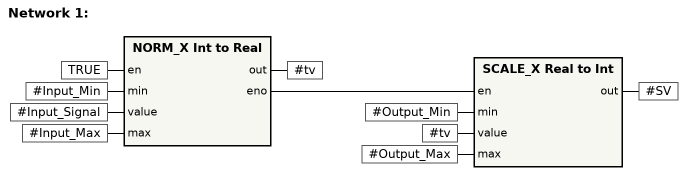
   IF TRUE THEN
       #tv := NORM_X(MIN := #Input_Min, VALUE := #Input_Signal, MAX := #Input_Max);
       #SV := SCALE_X(MIN := #Output_Min, VALUE := #tv, MAX := #Output_Max);
   END_IF;
END_REGION
END_FUNCTION

FUNCTION "CONVERTTIME" : Void   // FC2, FBD
{ S7_Optimized_Access := 'TRUE' }
VERSION : 0.1
   VAR_INPUT
      Int1 : Int;
   END_VAR
   VAR_OUTPUT
      tem1 : Time;
   END_VAR
   VAR_TEMP
      tv : Int;
   END_VAR
BEGIN

REGION Network 1
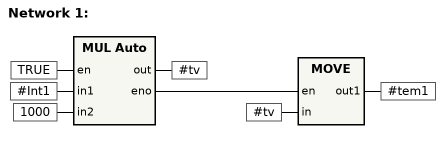
   IF TRUE THEN
       #tv := #Int1 * 1000;
       #tem1 := #tv;
   END_IF;
END_REGION
END_FUNCTION

ORGANIZATION_BLOCK "Main"   // OB1, LAD, ProgramCycle
TITLE = "Main Program Sweep (Cycle)"
{ S7_Optimized_Access := 'TRUE' }
VERSION : 0.1
   VAR_INPUT
      Initial_Call : Bool;   // Initial call of this OB
      Remanence : Bool;   // =True, if remanent data are available
   END_VAR
   VAR_TEMP
      InitiateSequens : Bool;
   END_VAR
   VAR_TEMP   // added for the SCL form of the ladder/FBD networks
      _w1 : Bool;
      _w2 : Bool;
      _w3 : Bool;
      _w4 : Bool;
   END_VAR
BEGIN

REGION Network 1
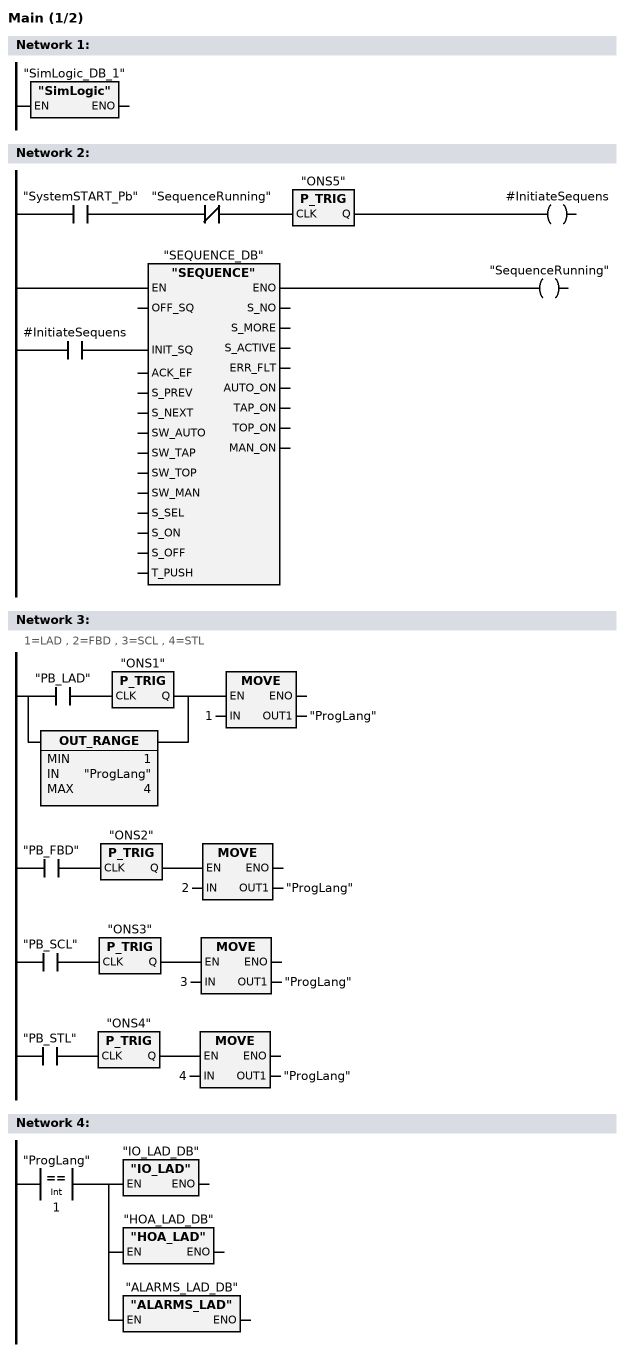
   RUNG wire#powerrail
      "SimLogic_DB_1"()
   END_RUNG
   // the same network as SCL:
   "SimLogic_DB_1"();   // "SimLogic"
END_REGION

REGION Network 2
   RUNG wire#powerrail
      Contact( "SystemSTART_Pb" )
      I_Contact( "SequenceRunning" )
      P_Trig( "ONS5" )
      Coil( #InitiateSequens )
   END_RUNG
   RUNG wire#powerrail
      "SEQUENCE_DB"(INIT_SQ := wire#w1, OFF_SQ :=, ACK_EF :=, S_PREV :=, S_NEXT :=, SW_AUTO :=, SW_TAP :=, SW_TOP :=, SW_MAN :=, S_SEL :=, S_ON :=, S_OFF :=, T_PUSH :=, S_NO =>, S_MORE =>, S_ACTIVE =>, ERR_FLT =>, AUTO_ON =>, TAP_ON =>, TOP_ON =>, MAN_ON =>)
      Coil( "SequenceRunning" )
   END_RUNG
   RUNG wire#powerrail
      Contact( #InitiateSequens )
   END_RUNG wire#w1
   // the same network as SCL:
   #_w1 := "SystemSTART_Pb" AND NOT "SequenceRunning";
   #_w2 := #_w1 AND NOT "ONS5";   // rising edge
   "ONS5" := #_w1;
   #InitiateSequens := #_w2;
   "SEQUENCE_DB"(INIT_SQ := #InitiateSequens, ENO => #_w3);   // "SEQUENCE"
   "SequenceRunning" := #_w3;
END_REGION

REGION Network 3
   // 1=LAD , 2=FBD , 3=SCL , 4=STL
   #_w1 := "PB_LAD" AND NOT "ONS1";   // rising edge
   "ONS1" := "PB_LAD";
   IF #_w1 OR ("ProgLang" < 1) OR ("ProgLang" > 4) THEN "ProgLang" := 1; END_IF;
   #_w2 := "PB_FBD" AND NOT "ONS2";   // rising edge
   "ONS2" := "PB_FBD";
   IF #_w2 THEN "ProgLang" := 2; END_IF;
   #_w3 := "PB_SCL" AND NOT "ONS3";   // rising edge
   "ONS3" := "PB_SCL";
   IF #_w3 THEN "ProgLang" := 3; END_IF;
   #_w4 := "PB_STL" AND NOT "ONS4";   // rising edge
   "ONS4" := "PB_STL";
   IF #_w4 THEN "ProgLang" := 4; END_IF;
END_REGION

REGION Network 4
   RUNG wire#powerrail
      { S7_Templates := "SrcType := Int" } EQ_Contact(in1 := "ProgLang", in2 := 1)
      wire#w1
      "IO_LAD_DB"()
   END_RUNG
   RUNG wire#w1
      "HOA_LAD_DB"()
   END_RUNG
   RUNG wire#w1
      "ALARMS_LAD_DB"()
   END_RUNG
   // the same network as SCL:
   #_w1 := "ProgLang" = 1;
   IF #_w1 THEN
       "IO_LAD_DB"();   // "IO_LAD"
       "HOA_LAD_DB"();   // "HOA_LAD"
       "ALARMS_LAD_DB"();   // "ALARMS_LAD"
   END_IF;
END_REGION

REGION Network 5
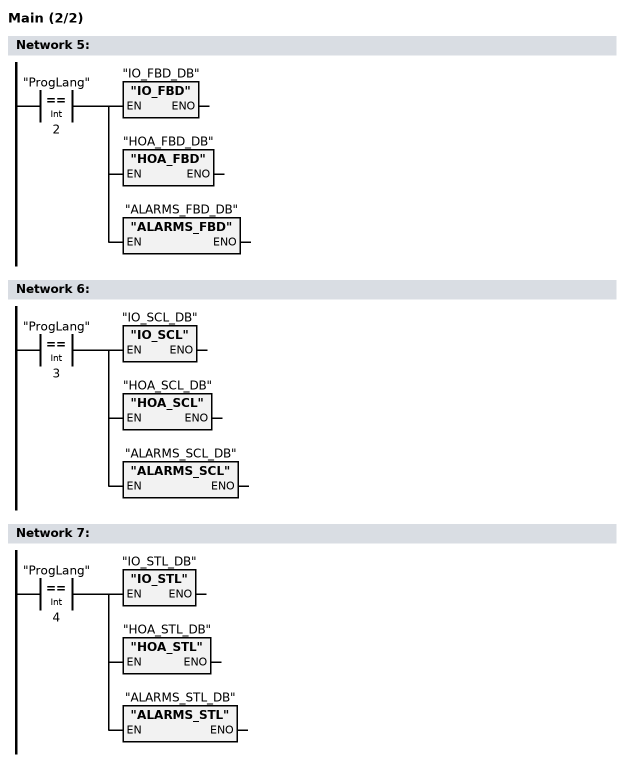
   RUNG wire#powerrail
      { S7_Templates := "SrcType := Int" } EQ_Contact(in1 := "ProgLang", in2 := 2)
      wire#w1
      "IO_FBD_DB"()
   END_RUNG
   RUNG wire#w1
      "HOA_FBD_DB"()
   END_RUNG
   RUNG wire#w1
      "ALARMS_FBD_DB"()
   END_RUNG
   // the same network as SCL:
   #_w1 := "ProgLang" = 2;
   IF #_w1 THEN
       "IO_FBD_DB"();   // "IO_FBD"
       "HOA_FBD_DB"();   // "HOA_FBD"
       "ALARMS_FBD_DB"();   // "ALARMS_FBD"
   END_IF;
END_REGION

REGION Network 6
   RUNG wire#powerrail
      { S7_Templates := "SrcType := Int" } EQ_Contact(in1 := "ProgLang", in2 := 3)
      wire#w1
      "IO_SCL_DB"()
   END_RUNG
   RUNG wire#w1
      "HOA_SCL_DB"()
   END_RUNG
   RUNG wire#w1
      "ALARMS_SCL_DB"()
   END_RUNG
   // the same network as SCL:
   #_w1 := "ProgLang" = 3;
   IF #_w1 THEN
       "IO_SCL_DB"();   // "IO_SCL"
       "HOA_SCL_DB"();   // "HOA_SCL"
       "ALARMS_SCL_DB"();   // "ALARMS_SCL"
   END_IF;
END_REGION

REGION Network 7
   RUNG wire#powerrail
      { S7_Templates := "SrcType := Int" } EQ_Contact(in1 := "ProgLang", in2 := 4)
      wire#w1
      "IO_STL_DB"()
   END_RUNG
   RUNG wire#w1
      "HOA_STL_DB"()
   END_RUNG
   RUNG wire#w1
      "ALARMS_STL_DB"()
   END_RUNG
   // the same network as SCL:
   #_w1 := "ProgLang" = 4;
   IF #_w1 THEN
       "IO_STL_DB"();   // "IO_STL"
       "HOA_STL_DB"();   // "HOA_STL"
       "ALARMS_STL_DB"();   // "ALARMS_STL"
   END_IF;
END_REGION
END_ORGANIZATION_BLOCK